FUNCTION_BLOCK FB_Ecat_State
VAR_INPUT
END_VAR

VAR
	raw_state AT %I* : ST_Ecat_State;
END_VAR

PROPERTY State : BOOL
GET
State := (NOT raw_state.wc_state) AND raw_state.op_state.3;
END_GET
END_PROPERTY

END_FUNCTION_BLOCK

(* stored: Version 1.1.0.1, ProductVersion 3.1.4024.12
   POU FB_Ecat_State: Id {15eb47f6-0c63-44c2-8753-ebab76c85955}, SpecialFunc None
   Property State: Id {a16b8eae-3f26-4062-a6b6-677f3643603f}
   Get Get: Id {3e8275b3-c530-4923-9995-e26764597daa} *)
